PROGRAM MAIN
VAR
END_VAR

IF Inputs.bEnableSimulation THEN
	CraneSimulation();
END_IF

END_PROGRAM

(* stored: Version 1.1.0.1, ProductVersion 3.1.4024.9
   POU MAIN: Id {a44625ec-42e1-4cf6-858d-5725a61c9069}, SpecialFunc None *)
